RoboDK station: test.rdk

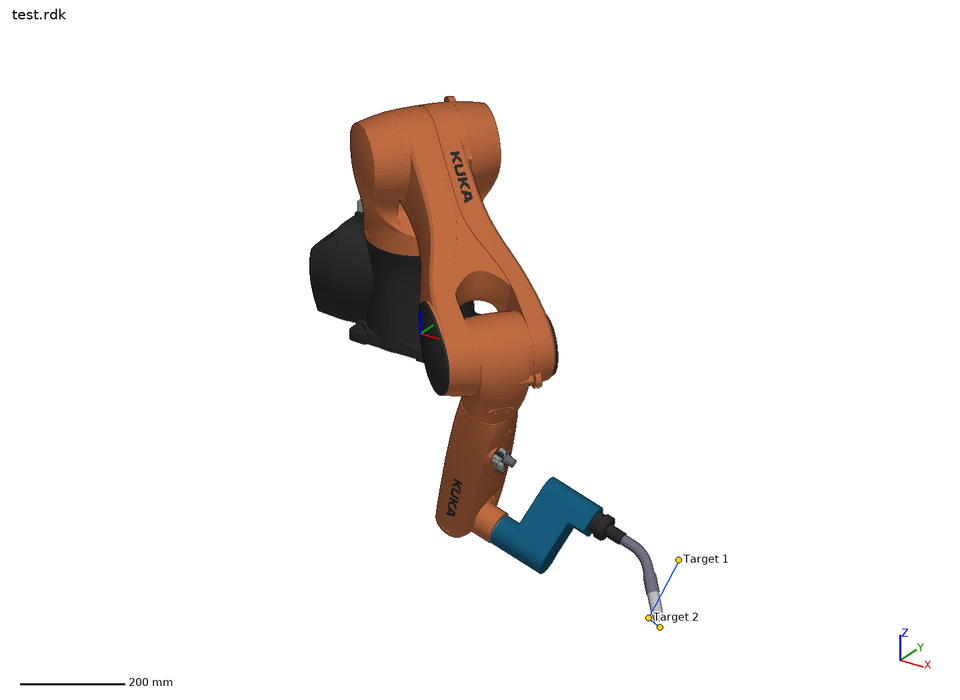
[picture v0: the station drawn from its stored meshes, robots at their saved joint values, targets as dots, program paths as lines]
Station test. Poses are relative to the parent item; angles as X-Y-Z fixed-axis rotations.
  - frame KUKA KR 10 R900 sixx Base at (0, 0, 0) mm
    - robot KUKA KR 10 R900 sixx: 6 axes, payload 10 kg, reach 901 mm, repeatability 0.03 mm, weight 52 kg
        modified DH rows (alpha deg, a mm, theta deg, d mm): 0, 0, 0, 400; -90, 25, 0, 0; 0, 455, -90, 0; -90, 35, 0, 420; 90, 0, 0, 0; -90, 0, 180, 80
        joint limits [-170, -190, -120, -185, -120, -350] to [170, 45, 156, 185, 120, 350]; home [0, -90, 90, 0, 0, 0]; saved at [35.062, 34.664, 80.583, 37.767, -89.173, 53.562]
      - tool Weld gun, TCP at (-4, 0, 371.3) mm, rotated rx 0 ry 45 rz 0 deg, size 299.9 x 60 x 318.3 mm
  - frame Frame 2 at (520.77, -1219.76, -366.26) mm, rotated rx -34.65 ry 0 rz 20.74 deg
    - target Target 1 (Cartesian target) at (492.81, 952.18, 685.28) mm, rotated rx -180 ry 19.81 rz -180 deg; joints [24.297, -46.747, 93.447, 50.375, -28.908, -35.715] of KUKA KR 10 R900 sixx
    - target Target 2 (Cartesian target) at (496.46, 748.35, 539.19) mm, rotated rx -180 ry 19.81 rz 180 deg; joints [38.326, -23.399, 69.264, -110.792, 36.887, 133.993] of KUKA KR 10 R900 sixx
    - target Target 3 (Cartesian target) at (496.46, 854.8, 539.19) mm, rotated rx -180 ry 19.81 rz 180 deg; joints [31.467, -29.133, 82.857, -128.099, 36.886, 149.032] of KUKA KR 10 R900 sixx
  - program Prog1 (5 instructions, listed below)
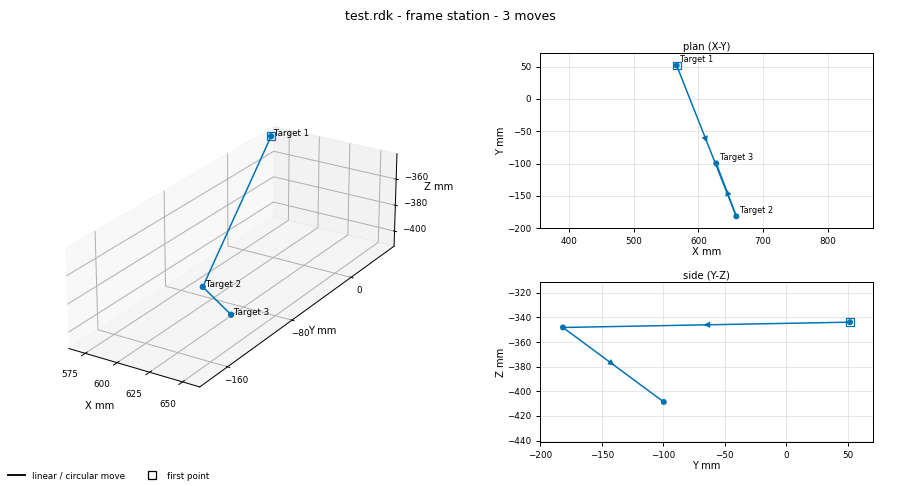
[picture p0: tool path of test.rdk in frame station, 3 of 3 moves have a stored position in this frame; points joined in program order, loops and branches not executed]

--- program Prog1 (robot KUKA KR 10 R900 sixx) ---
  Set Ref.: Frame 2
  Set Tool: Weld gun
  MoveJ (Target 1)
  MoveL (Target 2)
  MoveL (Target 3)
